// TIA Portal V19 export
DATA_BLOCK "PLCGlobal_DB"   // DB3
{ S7_Optimized_Access := 'TRUE' }
// stored: MemoryReserve 100
   VAR
      SafetyAckReset : Bool;
      GreenLampProcessActive : Bool;
      BluePushButton : Bool;
      SelectorSwitch : Bool;
      RedPushButton : Bool;
      GreenPushButtonLamp : Bool;
      BluePushButtonLamp : Bool;
      SelectorSwitchLamp : Bool;
      RedPushButtonLamp : Bool;
   END_VAR
BEGIN
END_DATA_BLOCK
